// TIA Portal project "PLC_stage_PREDIPLOMA" (V19)

(* hardware
DEVICE "S7-1500/ET200MP station_1"  S7-1500 station
   slot 0: "Rail_0"  Rack  6ES7 590-1***0-0AA0
   slot 1: "PLC_1"  CPU 1513F-1 PN  6ES7 513-1FL02-0AB0  V2.9
      slot 3: "CPU display_1"  6ES7591-1AA00-0AA0
      slot 32768: "PROFINET interface_1"  X1
      slot 34817: "Virtual CP interface port_1"  Virtual CP interface port  Virtual CP interface port
   slot 2: "DI 32x24VDC HF_1"  DI 32x24VDC HF  6ES7 521-1BL00-0AB0  V2.2
   slot 3: "DQ 32x24VDC/0.5A HF_1"  DQ 32x24VDC/0.5A HF  6ES7 522-1BL01-0AB0  V1.1
   slot 4: "AI 8xU/I/RTD/TC ST_1"  AI 8xU/I/RTD/TC ST  6ES7 531-7KF00-0AB0  V2.2
DEVICE "ET 200SP station_1"  ET 200SP-Station
   slot 0: "Rack_0"  Rack  6ES5 710-8MAx1
   slot 0: "IO device_1"  IM 155-6 PN ST  6ES7 155-6AU01-0BN0  V4.2
   slot 1: "DI 8x24VDC ST_1"  DI 8x24VDC ST  6ES7 131-6BF01-0BA0  V0.0
      slot 1: "DI 8x24VDC ST_1"  DI 8x24VDC ST
   slot 2: "DI 8x24VDC ST_2"  DI 8x24VDC ST  6ES7 131-6BF01-0BA0  V0.0
      slot 1: "DI 8x24VDC ST_2"  DI 8x24VDC ST
   slot 3: "DQ 16x24VDC/0.5A ST_1"  DQ 16x24VDC/0.5A ST  6ES7 132-6BH01-0BA0  V0.0
      slot 1: "DQ 16x24VDC/0.5A ST_1"  DQ 16x24VDC/0.5A ST
   slot 4: "AI 4xU/I 2-wire ST_2"  AI 4xU/I 2-wire ST  6ES7 134-6HD01-0BA1  V2.0
      slot 1: "AI 4xU/I 2-wire ST_2"  AI 4xU/I 2-wire ST
   slot 5: "AQ 4xU/I ST_1"  AQ 4xU/I ST  6ES7 135-6HD00-0BA1  V1.1
      slot 1: "AQ 4xU/I ST_1"  AQ 4xU/I ST
   slot 6: "Server module_1"  Server module  6ES7 193-6PA00-0AA0  V1.1
      slot 1: "Server module_1"  Server module
   slot 127: "BA 2xRJ45"  BA 2xRJ45  6ES7 193-6AR00-0AA0  V0.0
      slot 1: "Port_1"  X1 P1 R  6ES7 193-6AR00-0AA0  V0.0
      slot 2: "Port_2"  X1 P2 R  6ES7 193-6AR00-0AA0  V0.0
DEVICE "PC-System_1"  SIMATIC PC station
   slot 0: "SIMATIC PC station"  Rail  SIMATIC PC-Station  V1.0
      slot 125: "Stationmanager"  Station_Manager  V6.0.4
   slot 1: "HMI_RT_2"  WinCC RT Advanced  6AV2 104-0xxxx-xxxx  17.0.0.0
      slot 33792: "Computer interface"  Host interface
   slot 2: "IE general_1"  IE General  IE_CP  V8.2.0
      slot 1: "PROFINET interface"  IEGeneral.Interface.8.2.0
*)

// ===== PLC "PLC_1"  CPU 1513F-1 PN =====

VAR_GLOBAL   // PLC tag table "Default tag table"
   "Tag_2" AT %I20.0 : Bool;
   "Tag_3" AT %I20.1 : Bool;
   "Tag_4" AT %I20.2 : Bool;
   "Sensor1" AT %I29.0 : Bool;
   "Sensor2" AT %I29.1 : Bool;
   "Sensor3" AT %I29.2 : Bool;
   "Sensor4" AT %I29.3 : Bool;
   "System_Byte(1)" AT %MB1 : Byte;
   "Tag_1" AT %M11.0 : Bool;
   "Tag_5" AT %M11.1 : Bool;
END_VAR

VAR_GLOBAL   // PLC tag table "Default tag table_1"
   "sw1" AT %I0.0 : Bool;
   "sw2" AT %I0.1 : Bool;
   "sw3" AT %I0.2 : Bool;
   "sw4" AT %I0.3 : Bool;
   "Manip1" AT %Q0.0 : Bool;
   "K1" AT %Q4.0 : Bool;
   "Manip2" AT %Q0.2 : Bool;
   "FAN" AT %M11.3 : Bool;
   "amount" AT %MW1 : Int;
   "Manip1_counter" AT %MW2 : Int;
   "painting" AT %I1.1 : Bool;
   "tag1" AT %Q1.1 : Bool;
   "tag2" AT %Q1.2 : Bool;
   "Tag_1(1)" AT %T0 : Timer;
   "Tag_2(1)" AT %T1 : Timer;
   "pos1" AT %M1.3 : Bool;
   "pos2" AT %Q1.4 : Bool;
   "pos3" AT %M1.5 : Bool;
   "block_move" AT %MW4 : Int;
   "block_color" AT %Q1.6 : Bool;
   "start" AT %M6.0 : Bool;
   "stop" AT %M6.1 : Bool;
   "emergency" AT %M6.2 : Bool;
   "auto" AT %M6.3 : Bool;
   "manu" AT %M6.4 : Bool;
   "Tag_3(1)" AT %T2 : Timer;
   "Tag_4(1)" AT %T3 : Timer;
   "tag3" AT %M4.0 : Bool;
   "tag4" AT %M6.5 : Bool;
   "reset_block_pos" AT %M6.6 : Bool;
   "Clock_1.25Hz" AT %M0.4 : Bool;
   "Clock_1Hz" AT %M0.5 : Bool;
   "Clock_0.625Hz" AT %M0.6 : Bool;
   "Clock_0.5Hz" AT %M0.7 : Bool;
   "clocckk" AT %M3.0 : Bool;
   "manip_go_back" AT %M6.7 : Bool;
   "manip_cycle" AT %M3.1 : Bool;
   "p1" AT %M7.0 : Bool;
   "System_Byte" AT %MB0 : Byte;
   "FirstScan" AT %M0.0 : Bool;
   "DiagStatusUpdate" AT %M0.1 : Bool;
   "AlwaysTRUE" AT %M0.2 : Bool;
   "AlwaysFALSE" AT %M0.3 : Bool;
   "reset_manip_pos" AT %M21.0 : Bool;
   "Alarm_Collection" AT %MW21 : Int;
   "conv_error" AT %M24.0 : Bool;
   "manip1_error" AT %M24.1 : Bool;
   "manip2_error" AT %M24.2 : Bool;
   "fan_error" AT %M24.3 : Bool;
   "conv_broken" AT %M24.4 : Bool;
   "manip1_broken" AT %M24.5 : Bool;
   "manip2_broken" AT %M24.6 : Bool;
   "fan_broken" AT %M24.7 : Bool;
   "Tag_5(1)" AT %M12.0 : Bool;
END_VAR

VAR_GLOBAL CONSTANT   // PLC tag table "Default tag table_1"
   "None(1)" : Pip := 65535;
   "Automatic update(1)" : Pip := 0;
   "PIP 1(1)" : Pip := 1;
   "PIP 2(1)" : Pip := 2;
   "PIP 3(1)" : Pip := 3;
   "PIP 4(1)" : Pip := 4;
   "PIP 5(1)" : Pip := 5;
   "PIP 6(1)" : Pip := 6;
   "PIP 7(1)" : Pip := 7;
   "PIP 8(1)" : Pip := 8;
   "PIP 9(1)" : Pip := 9;
   "PIP 10(1)" : Pip := 10;
   "PIP 11(1)" : Pip := 11;
   "PIP 12(1)" : Pip := 12;
   "PIP 13(1)" : Pip := 13;
   "PIP 14(1)" : Pip := 14;
   "PIP 15(1)" : Pip := 15;
   "PIP 16(1)" : Pip := 16;
   "PIP 17(1)" : Pip := 17;
   "PIP 18(1)" : Pip := 18;
   "PIP 19(1)" : Pip := 19;
   "PIP 20(1)" : Pip := 20;
   "PIP 21(1)" : Pip := 21;
   "PIP 22(1)" : Pip := 22;
   "PIP 23(1)" : Pip := 23;
   "PIP 24(1)" : Pip := 24;
   "PIP 25(1)" : Pip := 25;
   "PIP 26(1)" : Pip := 26;
   "PIP 27(1)" : Pip := 27;
   "PIP 28(1)" : Pip := 28;
   "PIP 29(1)" : Pip := 29;
   "PIP 30(1)" : Pip := 30;
   "PIP 31(1)" : Pip := 31;
   "PIP OB Servo(1)" : Pip := 32768;
   "Local~MC(1)" : Hw_SubModule := 51;
   "Local~Common(1)" : Hw_SubModule := 50;
   "Local~Device(1)" : Hw_Device := 32;
   "Local~Configuration(1)" : Hw_SubModule := 33;
   "Local~Display(1)" : Hw_SubModule := 54;
   "Local~Exec(1)" : Hw_SubModule := 52;
   "Local(1)" : Hw_SubModule := 49;
   "Local~FExec(1)" : Hw_SubModule := 55;
   "Local~PROFINET_interface_1(1)" : Hw_Interface := 64;
   "Local~PROFINET_interface_1~Port_1(1)" : Hw_Interface := 65;
   "Local~PROFINET_interface_1~Port_2(1)" : Hw_Interface := 66;
   "Local~Virtual_communication_interface(1)" : Hw_Interface := 135;
   "Local~License_Manager(1)" : Hw_SubModule := 42;
   "OB_Main(1)" : OB_PCYCLE := 1;
   "OB_FOB_RTG1" : OB_Cyclic := 123;
   "Local~DI_32x24VDC_HF_1(1)" : Hw_SubModule := 257;
   "Local~DQ_32x24VDC_0_5A_HF_1(1)" : Hw_SubModule := 258;
   "Local~AI_8xU_I_HS_1" : Hw_SubModule := 259;
   "Local~AQ_8xU_I_HS_1" : Hw_SubModule := 260;
END_VAR

DATA_BLOCK "Block_1_DB"   // DB12
{ S7_Optimized_Access := 'TRUE' }
VERSION : 0.1
// stored: InstanceOfName Auto_mode
"Auto_mode"
BEGIN
END_DATA_BLOCK

DATA_BLOCK "Manu_mode_DB"   // DB13
{ S7_Optimized_Access := 'TRUE' }
VERSION : 0.1
// stored: InstanceOfName Manu_mode
"Manu_mode"
BEGIN
END_DATA_BLOCK

// folder: System blocks/Program resources

DATA_BLOCK "IEC_Counter_0_DB_3"   // DB2
{ S7_Optimized_Access := 'TRUE' }
AUTHOR : Simatic
FAMILY : IEC
NAME : CNTR
VERSION : 1.0
// stored: InstanceOfName IEC_COUNTER
"IEC_COUNTER"
BEGIN
END_DATA_BLOCK

DATA_BLOCK "IEC_Timer_0_DB_3"   // DB3
{ S7_Optimized_Access := 'TRUE' }
AUTHOR : Simatic
FAMILY : IEC
NAME : IEC_TMR
VERSION : 1.0
// stored: InstanceOfName IEC_TIMER
"IEC_TIMER"
BEGIN
END_DATA_BLOCK

DATA_BLOCK "IEC_Timer_0_DB"   // DB4
{ S7_Optimized_Access := 'TRUE' }
AUTHOR : Simatic
FAMILY : IEC
NAME : IEC_TMR
VERSION : 1.0
// stored: InstanceOfName IEC_TIMER
"IEC_TIMER"
BEGIN
END_DATA_BLOCK

DATA_BLOCK "IEC_Counter_0_DB_1"   // DB5
{ S7_Optimized_Access := 'TRUE' }
AUTHOR : Simatic
FAMILY : IEC
NAME : CNTR
VERSION : 1.0
// stored: InstanceOfName IEC_COUNTER
"IEC_COUNTER"
BEGIN
END_DATA_BLOCK

DATA_BLOCK "IEC_Timer_0_DB_1"   // DB6
{ S7_Optimized_Access := 'TRUE' }
AUTHOR : Simatic
FAMILY : IEC
NAME : IEC_TMR
VERSION : 1.0
// stored: InstanceOfName IEC_TIMER
"IEC_TIMER"
BEGIN
END_DATA_BLOCK

DATA_BLOCK "IEC_Timer_0_DB_2"   // DB7
{ S7_Optimized_Access := 'TRUE' }
AUTHOR : Simatic
FAMILY : IEC
NAME : IEC_TMR
VERSION : 1.0
// stored: InstanceOfName IEC_TIMER
"IEC_TIMER"
BEGIN
END_DATA_BLOCK

DATA_BLOCK "IEC_Timer_0_DB_5"   // DB8
{ S7_Optimized_Access := 'TRUE' }
AUTHOR : Simatic
FAMILY : IEC
NAME : IEC_TMR
VERSION : 1.0
// stored: InstanceOfName IEC_TIMER
"IEC_TIMER"
BEGIN
END_DATA_BLOCK

DATA_BLOCK "IEC_Timer_0_DB_6"   // DB9
{ S7_Optimized_Access := 'TRUE' }
AUTHOR : Simatic
FAMILY : IEC
NAME : IEC_TMR
VERSION : 1.0
// stored: InstanceOfName IEC_TIMER
"IEC_TIMER"
BEGIN
END_DATA_BLOCK

DATA_BLOCK "IEC_Timer_0_DB_4"   // DB10
{ S7_Optimized_Access := 'TRUE' }
AUTHOR : Simatic
FAMILY : IEC
NAME : IEC_TMR
VERSION : 1.0
// stored: InstanceOfName IEC_TIMER
"IEC_TIMER"
BEGIN
END_DATA_BLOCK

DATA_BLOCK "IEC_Counter_0_DB_2"   // DB11
{ S7_Optimized_Access := 'TRUE' }
AUTHOR : Simatic
FAMILY : IEC
NAME : CNTR
VERSION : 1.0
// stored: InstanceOfName IEC_COUNTER
"IEC_COUNTER"
BEGIN
END_DATA_BLOCK

// folder: (top level)

FUNCTION_BLOCK "Auto_mode"   // FB2, LAD
{ S7_Optimized_Access := 'TRUE' }
VERSION : 0.1
   VAR_TEMP   // added for the SCL form of the ladder/FBD networks
      _w1 : Bool;
      _w2 : Bool;
      _w3 : Bool;
      _w4 : Bool;
   END_VAR
BEGIN

REGION Network 1
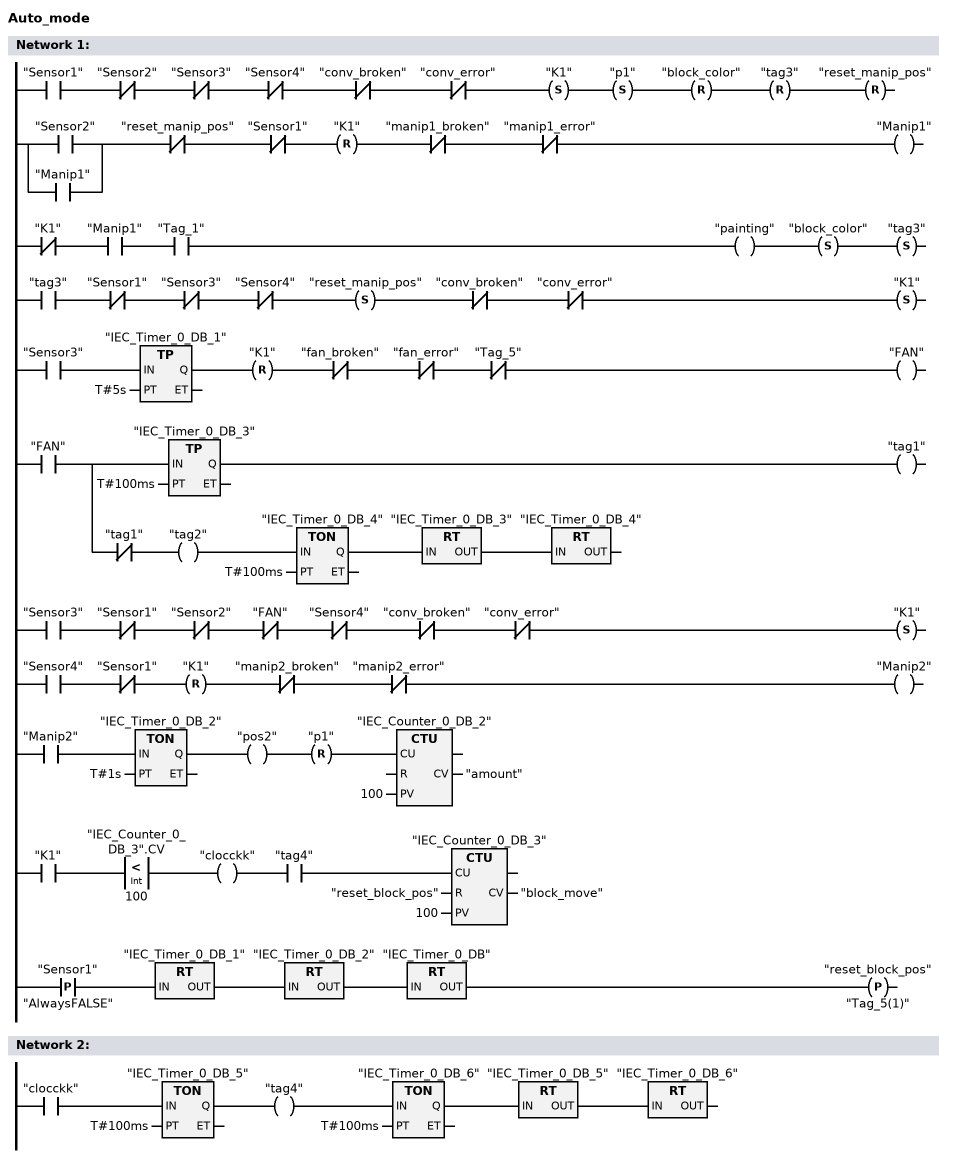
   IF "Sensor1" AND NOT "Sensor2" AND NOT "Sensor3" AND NOT "Sensor4" AND NOT "conv_broken" AND NOT "conv_error" THEN
       "K1" := TRUE;
       "p1" := TRUE;
       "block_color" := FALSE;
       "tag3" := FALSE;
       "reset_manip_pos" := FALSE;
   END_IF;
   #_w1 := ("Sensor2" OR "Manip1") AND NOT "reset_manip_pos" AND NOT "Sensor1";
   IF #_w1 THEN "K1" := FALSE; END_IF;
   "Manip1" := #_w1 AND NOT "manip1_broken" AND NOT "manip1_error";
   "painting" := NOT "K1" AND "Manip1" AND "Tag_1";
   IF "painting" THEN
       "block_color" := TRUE;
       "tag3" := TRUE;
   END_IF;
   #_w2 := "tag3" AND NOT "Sensor1" AND NOT "Sensor3" AND NOT "Sensor4";
   IF #_w2 THEN "reset_manip_pos" := TRUE; END_IF;
   IF #_w2 AND NOT "conv_broken" AND NOT "conv_error" THEN "K1" := TRUE; END_IF;
   "IEC_Timer_0_DB_1".TP(IN := "Sensor3", PT := T#5s);
   IF "IEC_Timer_0_DB_1".Q THEN "K1" := FALSE; END_IF;
   "FAN" := "IEC_Timer_0_DB_1".Q AND NOT "fan_broken" AND NOT "fan_error" AND NOT "Tag_5";
   "IEC_Timer_0_DB_3".TP(IN := "FAN", PT := T#100ms);
   "tag1" := "IEC_Timer_0_DB_3".Q;
   "tag2" := "FAN" AND NOT "tag1";
   "IEC_Timer_0_DB_4".TON(IN := "tag2", PT := T#100ms);
   IF "IEC_Timer_0_DB_4".Q THEN
       RESET_TIMER("IEC_Timer_0_DB_3");
       RESET_TIMER("IEC_Timer_0_DB_4");
   END_IF;
   IF "Sensor3" AND NOT "Sensor1" AND NOT "Sensor2" AND NOT "FAN" AND NOT "Sensor4" AND NOT "conv_broken" AND NOT "conv_error" THEN
       "K1" := TRUE;
   END_IF;
   #_w3 := "Sensor4" AND NOT "Sensor1";
   IF #_w3 THEN "K1" := FALSE; END_IF;
   "Manip2" := #_w3 AND NOT "manip2_broken" AND NOT "manip2_error";
   "IEC_Timer_0_DB_2".TON(IN := "Manip2", PT := T#1s);
   "pos2" := "IEC_Timer_0_DB_2".Q;
   IF "IEC_Timer_0_DB_2".Q THEN "p1" := FALSE; END_IF;
   "IEC_Counter_0_DB_2".CTU(CU := "IEC_Timer_0_DB_2".Q, PV := 100, CV => "amount");
   "clocckk" := "K1" AND ("IEC_Counter_0_DB_3".CV < 100);
   "IEC_Counter_0_DB_3".CTU(CU := "clocckk" AND "tag4", R := "reset_block_pos", PV := 100, CV => "block_move");
   #_w4 := "Sensor1" AND NOT "AlwaysFALSE";   // rising edge of "Sensor1"
   "AlwaysFALSE" := "Sensor1";
   IF #_w4 THEN
       RESET_TIMER("IEC_Timer_0_DB_1");
       RESET_TIMER("IEC_Timer_0_DB_2");
       RESET_TIMER("IEC_Timer_0_DB");
   END_IF;
   "reset_block_pos" := #_w4 AND NOT "Tag_5(1)";   // rising edge
   "Tag_5(1)" := #_w4;
END_REGION

REGION Network 2
   "IEC_Timer_0_DB_5".TON(IN := "clocckk", PT := T#100ms);
   "tag4" := "IEC_Timer_0_DB_5".Q;
   "IEC_Timer_0_DB_6".TON(IN := "IEC_Timer_0_DB_5".Q, PT := T#100ms);
   IF "IEC_Timer_0_DB_6".Q THEN
       RESET_TIMER("IEC_Timer_0_DB_5");
       RESET_TIMER("IEC_Timer_0_DB_6");
   END_IF;
END_REGION
END_FUNCTION_BLOCK

FUNCTION_BLOCK "Manu_mode"   // FB3, LAD
{ S7_Optimized_Access := 'TRUE' }
VERSION : 0.1
   VAR_TEMP   // added for the SCL form of the ladder/FBD networks
      _w1 : Bool;
      _w2 : Bool;
   END_VAR
BEGIN

REGION Network 1
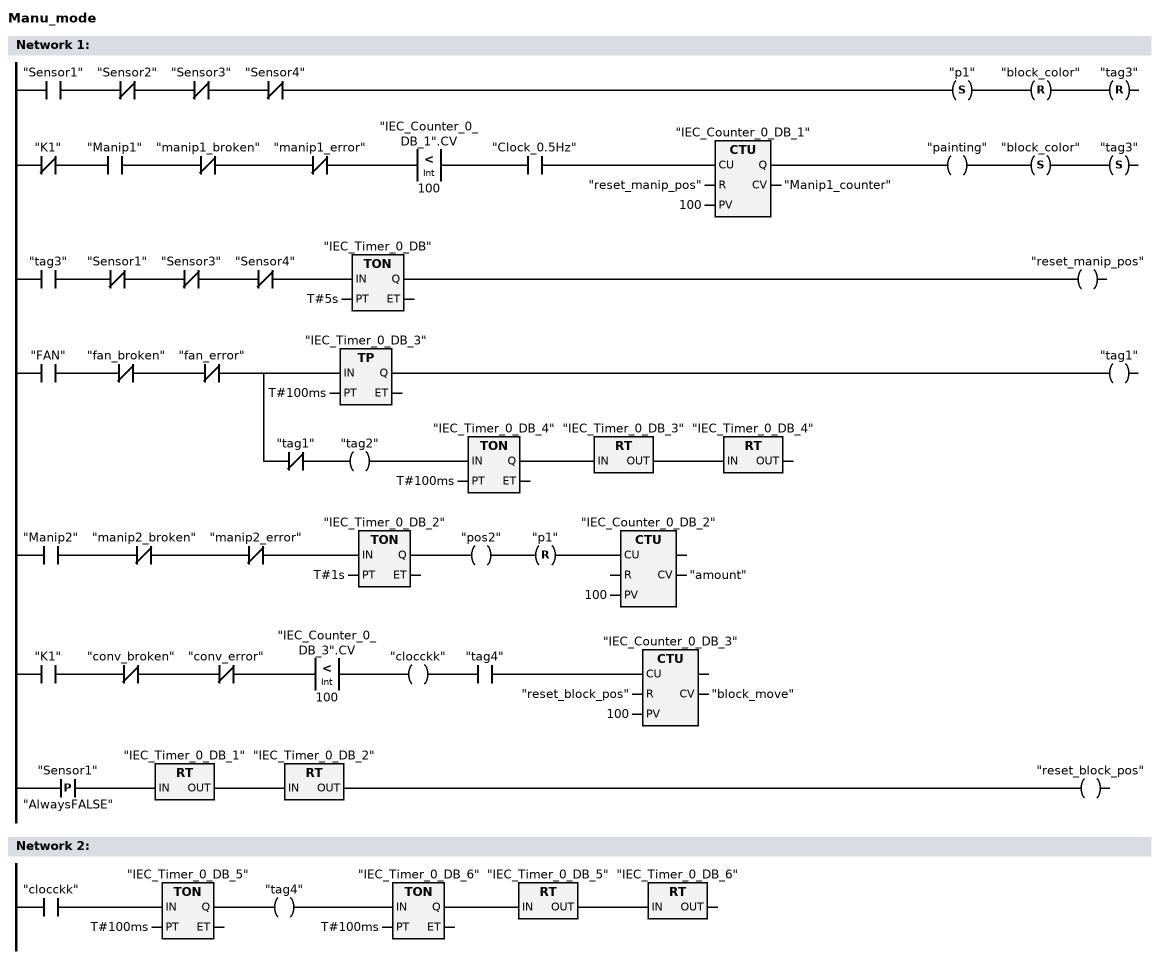
   IF "Sensor1" AND NOT "Sensor2" AND NOT "Sensor3" AND NOT "Sensor4" THEN
       "p1" := TRUE;
       "block_color" := FALSE;
       "tag3" := FALSE;
   END_IF;
   "IEC_Counter_0_DB_1".CTU(CU := NOT "K1" AND "Manip1" AND NOT "manip1_broken" AND NOT "manip1_error" AND ("IEC_Counter_0_DB_1".CV < 100) AND "Clock_0.5Hz",
                           R := "reset_manip_pos",
                           PV := 100,
                           CV => "Manip1_counter");
   "painting" := "IEC_Counter_0_DB_1".Q;
   IF "IEC_Counter_0_DB_1".Q THEN
       "block_color" := TRUE;
       "tag3" := TRUE;
   END_IF;
   "IEC_Timer_0_DB".TON(IN := "tag3" AND NOT "Sensor1" AND NOT "Sensor3" AND NOT "Sensor4", PT := T#5s);
   "reset_manip_pos" := "IEC_Timer_0_DB".Q;
   #_w1 := "FAN" AND NOT "fan_broken" AND NOT "fan_error";
   "IEC_Timer_0_DB_3".TP(IN := #_w1, PT := T#100ms);
   "tag1" := "IEC_Timer_0_DB_3".Q;
   "tag2" := #_w1 AND NOT "tag1";
   "IEC_Timer_0_DB_4".TON(IN := "tag2", PT := T#100ms);
   IF "IEC_Timer_0_DB_4".Q THEN
       RESET_TIMER("IEC_Timer_0_DB_3");
       RESET_TIMER("IEC_Timer_0_DB_4");
   END_IF;
   "IEC_Timer_0_DB_2".TON(IN := "Manip2" AND NOT "manip2_broken" AND NOT "manip2_error", PT := T#1s);
   "pos2" := "IEC_Timer_0_DB_2".Q;
   IF "IEC_Timer_0_DB_2".Q THEN "p1" := FALSE; END_IF;
   "IEC_Counter_0_DB_2".CTU(CU := "IEC_Timer_0_DB_2".Q, PV := 100, CV => "amount");
   "clocckk" := "K1" AND NOT "conv_broken" AND NOT "conv_error" AND ("IEC_Counter_0_DB_3".CV < 100);
   "IEC_Counter_0_DB_3".CTU(CU := "clocckk" AND "tag4", R := "reset_block_pos", PV := 100, CV => "block_move");
   #_w2 := "Sensor1" AND NOT "AlwaysFALSE";   // rising edge of "Sensor1"
   "AlwaysFALSE" := "Sensor1";
   IF #_w2 THEN
       RESET_TIMER("IEC_Timer_0_DB_1");
       RESET_TIMER("IEC_Timer_0_DB_2");
   END_IF;
   "reset_block_pos" := #_w2;
END_REGION

REGION Network 2
   "IEC_Timer_0_DB_5".TON(IN := "clocckk", PT := T#100ms);
   "tag4" := "IEC_Timer_0_DB_5".Q;
   "IEC_Timer_0_DB_6".TON(IN := "IEC_Timer_0_DB_5".Q, PT := T#100ms);
   IF "IEC_Timer_0_DB_6".Q THEN
       RESET_TIMER("IEC_Timer_0_DB_5");
       RESET_TIMER("IEC_Timer_0_DB_6");
   END_IF;
END_REGION
END_FUNCTION_BLOCK

ORGANIZATION_BLOCK "Main"   // OB1, LAD, ProgramCycle
TITLE = "Main Program Sweep (Cycle)"
{ S7_Optimized_Access := 'TRUE' }
VERSION : 0.1
   VAR_INPUT
      Initial_Call : Bool;   // Initial call of this OB
      Remanence : Bool;   // =True, if remanent data are available
   END_VAR
BEGIN

REGION Network 1
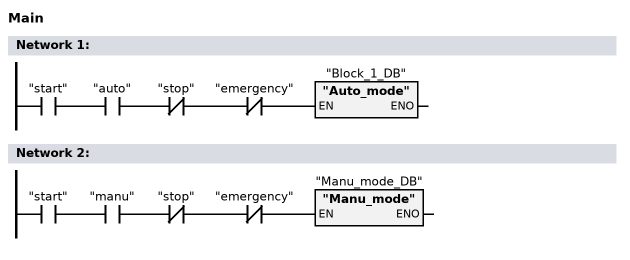
   RUNG wire#powerrail
      Contact( "start" )
      Contact( "auto" )
      I_Contact( "stop" )
      I_Contact( "emergency" )
      "Block_1_DB"()
   END_RUNG
   // the same network as SCL:
   IF "start" AND "auto" AND NOT "stop" AND NOT "emergency" THEN
       "Block_1_DB"();   // "Auto_mode"
   END_IF;
END_REGION

REGION Network 2
   RUNG wire#powerrail
      Contact( "start" )
      Contact( "manu" )
      I_Contact( "stop" )
      I_Contact( "emergency" )
      "Manu_mode_DB"()
   END_RUNG
   // the same network as SCL:
   IF "start" AND "manu" AND NOT "stop" AND NOT "emergency" THEN
       "Manu_mode_DB"();   // "Manu_mode"
   END_IF;
END_REGION
END_ORGANIZATION_BLOCK

// ===== PLC "PLC_2"   =====

(* ===== HMI "HMI_RT_2" =====
system functions are stored by id; their names below are inferred from use
connection "HMI_Connection_2": ETHERNET, S7_1500_OMS
connection "HMI_Connection_1": ETHERNET, S7_1500_OMS

HMI tags "Default tag table"
   "Manip1_counter" : Int = PLC Manip1_counter AT %MW2, 1 s
   "tag1" : Bool = PLC tag1 AT %Q1.1, 1 s
   "tag2" : Bool = PLC tag2 AT %Q1.2, 1 s
   "sw1" : Bool = PLC sw1 AT %I0.0, 1 s
   "sw2" : Bool = PLC sw2 AT %I0.1, 1 s
   "sw3" : Bool = PLC sw3 AT %I0.2, 1 s
   "sw4" : Bool = PLC sw4 AT %I0.3, 1 s
   "Manip1" : Bool = PLC Manip1 AT %Q0.0, 1 s
   "FAN" : Bool = PLC FAN AT %M11.3, 1 s
   "K1" : Bool = PLC K1 AT %Q0.1, 1 s
   "Manip2" : Bool = PLC Manip2 AT %Q0.2, 1 s
   "pos2" : Bool = PLC pos2 AT %Q1.4, 1 s
   "amount" : Int = PLC amount AT %MW1, 1 s
   "painting" : Bool = PLC painting AT %I1.1, 1 s
   "block_move" : Int = PLC block_move AT %MW4, 1 s
   "block_color" : Bool = PLC block_color AT %Q1.6, 1 s
   "start" : Bool = PLC start AT %M6.0, 1 s
   "IEC_Counter_0_DB_1_CV" : Int = PLC IEC_Counter_0_DB_1.CV, 1 s
   "p1" : Bool = PLC p1 AT %M7.0, 1 s
   "emergency" : Bool = PLC emergency AT %M6.2, 1 s
   "stop" : Bool = PLC stop AT %M6.1, 1 s
   "auto" : Bool = PLC auto AT %M6.3, 1 s
   "manu" : Bool = PLC manu AT %M6.4, 1 s
   "Alarm_Collection" : Int = PLC Alarm_Collection AT %MW21, 1 s
   "manip1_error" : Bool = PLC manip1_error AT %M24.1, 1 s
   "manip1_broken" : Bool = PLC manip1_broken AT %M24.5, 1 s
   "fan_error" : Bool = PLC fan_error AT %M24.3, 1 s
   "fan_broken" : Bool = PLC fan_broken AT %M24.7, 1 s
   "conv_broken" : Bool = PLC conv_broken AT %M24.4, 1 s
   "conv_error" : Bool = PLC conv_error AT %M24.0, 1 s
   "manip2_error" : Bool = PLC manip2_error AT %M24.2, 1 s
   "manip2_broken" : Bool = PLC manip2_broken AT %M24.6, 1 s

discrete alarms
   1: 'Something is wrong with the conveyor!!!', class Errors, trigger "Alarm_Collection" bit 0
   2: 'Conveyor is in tech-service.', class Warnings, trigger "Alarm_Collection" bit 1
   3: 'Something is wrong with the Manipulator 1!!!', class Errors, trigger "Alarm_Collection" bit 2
   4: 'Manipulator 1 is in tech-service.', class Warnings, trigger "Alarm_Collection" bit 3
   5: 'Something is wrong with the Fan!!!', class Errors, trigger "Alarm_Collection" bit 4
   6: 'Fan is in tech-service.', class Warnings, trigger "Alarm_Collection" bit 5
   7: 'Something is wrong with the Manipulator 2!!!', class Errors, trigger "Alarm_Collection" bit 6
   8: 'Manipulator 2 is in tech-service.', class Warnings, trigger "Alarm_Collection" bit 7

text list "OFF_ON_LIST": 0 ''; 1 ''

screen "Screen_2" 1980x1080
   Circle "Circle_6" at 216,721 size 41x41
      Appearance <- "Manip1"
   IOField "I/O field_1" at 1077,716 size 145x38; FormatPattern s99999
      ProcessValue <- "amount"
   Circle "Circle_7" at 1051,213 size 41x41
      Appearance <- "Manip2"
   TextField "Text field_1" at 225,778 size 210x70; Text 'MANIPULATOR Spray'
   TextField "Text field_2" at 590,707 size 60x37; Text 'FAN'
   TextField "Text field_3" at 1071,771 size 144x37; Text 'Packeging'
   TextField "Text field_4" at 1043,137 size 210x70; Text 'MANIPULATOR Pick & Place'
   TextField "Text field_6" at 140,158 size 41x39; Text 'S1'
   TextField "Text field_5" at 297,158 size 41x39; Text 'S2'
   TextField "Text field_7" at 452,158 size 41x39; Text 'S3'
   TextField "Text field_8" at 856,159 size 41x39; Text 'S4'
   Button "Button_2" at 1360,84 size 133x57; TextOff 'Start'; TextList "OFF_ON_LIST"
      on Press: SetBit("start"); ResetBit("stop")
      ProcessValue <- "start"
   Button "Button_6" at 1360,172 size 133x57; TextOff 'STOP'
      on Press: SetBit("stop"); ResetBit("start")
      on Release: ResetBit("stop")
      Visibility <- "stop"
   GraphicView "Graphic view_2" at 375,721 size 49x47; Picture "Graphic_7"
      Visibility <- "manip1_broken"
   GraphicView "Graphic view_3" at 293,721 size 49x47; Picture "Graphic_8"
      Visibility <- "manip1_error"
   GraphicView "Graphic view_5" at 1199,213 size 49x47; Picture "Graphic_7"
      Appearance <- "manip2_broken"
   GraphicView "Graphic view_7" at 1124,212 size 49x47; Picture "Graphic_8"
      Appearance <- "manip2_error"
   Circle "Circle_16" at 147,213 size 29x29
      Appearance <- "sw1"
   Circle "Circle_18" at 298,211 size 29x29
      Appearance <- "sw2"
   Circle "Circle_20" at 758,488 size 41x41
      Appearance <- "K1"
   GraphicView "Graphic view_1" at 832,488 size 49x47; Picture "Graphic_8"
      Appearance <- "conv_error"
   GraphicView "Graphic view_8" at 904,488 size 49x47; Picture "Graphic_7"
      Appearance <- "conv_broken"
   TextField "Text field_11" at 797,544 size 134x37; Text 'Conveyor'
   Circle "Circle_8" at 455,210 size 29x29
      Appearance <- "sw3"
   Circle "Circle_9" at 858,208 size 29x29
      Appearance <- "sw4"
   Rectangle "Rectangle_15" at 1100,329 size 76x141
      Visibility <- "pos2"
   Rectangle "Rectangle_18" at 1116,472 size 49x109
      Visibility <- "pos2"
   Rectangle "Rectangle_19" at 1109,580 size 64x24
      Visibility <- "pos2"
   Group "Group" at 128,304 size 110x99
      HorizontalMovement <- "block_move"
   Button "Button_8" at 1752,423 size 96x41; TextOff 'sw1'
      on Press: SetBit("sw1")
      on Release: ResetBit("sw1")
   Button "Button_9" at 1752,483 size 96x41; TextOff 'sw2'
      on Press: SetBit("sw2")
      on Release: ResetBit("sw2")
   Button "Button_10" at 1752,541 size 96x41; TextOff 'sw3'
      on Press: SetBit("sw3")
      on Release: ResetBit("sw3")
   Button "Button_11" at 1752,600 size 96x41; TextOff 'sw4'
      on Press: SetBit("sw4")
      on Release: ResetBit("sw4")
   Circle "Circle_12" at 296,320 size 47x47
      Visibility <- "painting"
   Rectangle "Rectangle_11" at 300,448 size 39x199
      VerticalMovement <- "IEC_Counter_0_DB_1_CV"
   Rectangle "Rectangle_12" at 294,426 size 49x23
      VerticalMovement <- "IEC_Counter_0_DB_1_CV"
   Circle "Circle_11" at 523,652 size 41x41
      Appearance <- "FAN"
   GraphicView "Graphic view_4" at 658,651 size 49x47; Picture "Graphic_7"
      Appearance <- "fan_broken"
   GraphicView "Graphic view_6" at 592,651 size 49x47; Picture "Graphic_8"
      Appearance <- "fan_error"
   GraphicView "Graphic view_9" at 551,197 size 129x125; Picture "Graphic_14"
      Visibility <- "FAN"
   GraphicView "Graphic view_10" at 551,198 size 129x125; Picture "Graphic_15"
      Visibility <- "tag1"
   Rectangle "Rectangle_22" at 1031,329 size 147x73
      Visibility <- "pos2"
   Rectangle "Rectangle_23" at 918,340 size 113x47
      Visibility <- "pos2"
   Rectangle "Rectangle_24" at 893,333 size 25x61
      Visibility <- "pos2"
   GraphicView "Graphic view_13" at 551,197 size 129x125; Picture "Graphic_16"
      Visibility <- "tag2"
   GraphicView "Graphic view_11" at 551,353 size 129x125; Picture "Graphic_14"
   GraphicView "Graphic view_12" at 551,353 size 129x125; Picture "Graphic_15"
      Visibility <- "tag1"
   GraphicView "Graphic view_14" at 551,353 size 129x125; Picture "Graphic_16"
      Visibility <- "tag2"
   Circle "Circle_13" at 36,54 size 90x90
      Appearance <- "emergency"
   Button "Button_12" at 1519,126 size 174x56; TextOff 'Emergency'
      on Press: SetBit("emergency"); ResetBit("start"); ResetBit("auto"); ResetBit("manu")
      on Release: ResetBit("emergency")
   Button "Button_1" at 1718,172 size 133x57; TextOff 'Auto Mode'
      on Press: SetBit("auto"); ResetBit("manu")
      Visibility <- "auto"
   Button "Button_13" at 1718,84 size 133x57; TextOff 'Manu Mode'
      on Press: SetBit("manu"); ResetBit("auto")
      Visibility <- "manu"
   Button "Button_14" at 1360,256 size 190x61; TextOff 'MANIPULATOR Spray'
      on Press: SetBit("Manip1")
      on Release: ResetBit("Manip1")
   Button "Button_3" at 1660,256 size 190x61; TextOff 'MANIPULATOR Pick & Place'
      on Press: SetBit("Manip2")
      on Release: ResetBit("Manip2")
   Button "Button_4" at 1360,338 size 190x61; TextOff 'FAN'
      on Press: SetBit("FAN")
      on Release: ResetBit("FAN")
   Button "Button_5" at 1660,338 size 190x61; TextOff 'Conveyor'
      on Press: SetBit("K1")
      on Release: ResetBit("K1")
   AlarmView "Alarm view_1" at 1360,754 size 499x232
   TextField "Text field_9" at 1513,712 size 190x33; Text 'ERROR STATUS'
   TextField "Text field_10" at 1507,25 size 209x33; Text 'CONTROL PANEL'
   GraphicView "Graphic view_15" at 293,721 size 49x47; Picture "Graphic_10"
      Visibility <- "manip1_error"
   GraphicView "Graphic view_16" at 375,721 size 49x47; Picture "Graphic_9"
      Visibility <- "manip1_broken"
   GraphicView "Graphic view_17" at 592,651 size 49x47; Picture "Graphic_10"
      Visibility <- "fan_error"
   GraphicView "Graphic view_18" at 658,651 size 49x47; Picture "Graphic_9"
      Visibility <- "fan_broken"
   GraphicView "Graphic view_19" at 904,488 size 49x47; Picture "Graphic_9"
      Visibility <- "conv_broken"
   GraphicView "Graphic view_20" at 832,488 size 49x47; Picture "Graphic_10"
      Visibility <- "conv_error"
   GraphicView "Graphic view_21" at 1124,212 size 49x47; Picture "Graphic_10"
      Visibility <- "manip2_error"
   GraphicView "Graphic view_22" at 1199,213 size 49x47; Picture "Graphic_9"
      Visibility <- "manip2_broken"
   Button "Button_17" at 1360,423 size 180x43; TextOff 'Conv error'
      on Press: function_b3f726e6("Alarm_Collection", 0); SetBit("conv_error")
   Button "Button_18" at 1360,473 size 180x43; TextOff 'Conv broken'
      on Press: function_b3f726e6("Alarm_Collection", 1); SetBit("conv_broken")
   Button "Button_20" at 1360,523 size 180x43; TextOff 'manip1 error'
      on Press: function_b3f726e6("Alarm_Collection", 2); SetBit("manip1_error")
   Button "Button_22" at 1360,573 size 180x43; TextOff 'manip1 broken'
      on Press: function_b3f726e6("Alarm_Collection", 3); SetBit("manip1_broken")
   Button "Button_19" at 1555,423 size 180x43; TextOff 'Fan error'
      on Press: function_b3f726e6("Alarm_Collection", 4); SetBit("fan_error")
   Button "Button_23" at 1555,473 size 180x43; TextOff 'Fan broken'
      on Press: function_b3f726e6("Alarm_Collection", 5); SetBit("fan_broken")
   Button "Button_24" at 1555,523 size 180x43; TextOff 'manip2 error'
      on Press: function_b3f726e6("Alarm_Collection", 6); SetBit("manip2_error")
   Button "Button_25" at 1555,573 size 180x43; TextOff 'manip2 broken'
      on Press: function_b3f726e6("Alarm_Collection", 7); SetBit("manip2_broken")
   Button "Button_7" at 1425,625 size 238x43; TextOff 'Repair all'
      on Press: function_a9b64e44("Alarm_Collection", 0); function_a9b64e44("Alarm_Collection", 1); function_a9b64e44("Alarm_Collection", 2); function_a9b64e44("Alarm_Collection", 3); function_a9b64e44("Alarm_Collection", 4); function_a9b64e44("Alarm_Collection", 5); function_a9b64e44("Alarm_Collection", 6); function_a9b64e44("Alarm_Collection", 7); ResetBit("conv_error"); ResetBit("conv_broken"); ResetBit("manip1_error"); ResetBit("manip1_broken"); ResetBit("fan_error"); ResetBit("fan_broken"); ResetBit("manip2_error"); ResetBit("manip2_broken")
   Rectangle "Rectangle_44" at 128,304 size 110x74
      Appearance <- "block_color"
      Visibility <- "p1"
   Rectangle "Rectangle_45" at 128,378 size 110x25
      Appearance <- "block_color"
      Visibility <- "p1"
*)